(* IEC 61131-3 sources: mp-conveyorbelt/test, 4 files *)

(* ---- ProcessStateAssert.st ---- *)
USING Simatic.Ax.Process;
USING AxUnit.ResultFunctions;
USING System.Strings;
USING Simatic.Ax.Process;

NAMESPACE AxUnit.Assert
    FUNCTION PUBLIC Equal
        VAR_INPUT
            actual : ProcessState;
            expected: ProcessState;
            {CallerFilePath}
            file : WSTRING[1024];
            {CallerLineNumber}
            line : INT;
        END_VAR

        IF actual = expected THEN
            axunit_Succeed();
        ELSE
            axunit_Fail('ProcessState assertion failed', file, line);
        END_IF;

    END_FUNCTION
END_NAMESPACE

(* ---- conveyorbelt-tests.st ---- *)
USING Simatic.Ax.Mp;

NAMESPACE SimaticAxMp

    {TestFixture}
    CLASS Test_SensorInfeed
        {Test}
        METHOD PUBLIC Test_x
            AxUnit.Assert.Equal(expected := 2, actual := 2);
        END_METHOD
        {Test}
        METHOD PUBLIC Test_y
            ; // AxUnit.Assert.Equal(expected := y, actual := x);
        END_METHOD
    END_CLASS

    {TestFixture}
    CLASS Test_SensorWork
        {Test}
        METHOD PUBLIC Test_x
            ; // AxUnit.Assert.Equal(expected := y, actual := x);
        END_METHOD
        {Test}
        METHOD PUBLIC Test_y
            ; // AxUnit.Assert.Equal(expected := y, actual := x);
        END_METHOD
    END_CLASS

    {TestFixture}
    CLASS Test_SensorOutfeed
        {Test}
        METHOD PUBLIC Test_x
            ; // AxUnit.Assert.Equal(expected := y, actual := x);
        END_METHOD
        {Test}
        METHOD PUBLIC Test_y
            ; // AxUnit.Assert.Equal(expected := y, actual := x);
        END_METHOD
    END_CLASS

    {TestFixture}
    CLASS Test_AxisControl
        {Test}
        METHOD PUBLIC Test_x
            ; // AxUnit.Assert.Equal(expected := y, actual := x);
        END_METHOD
        {Test}
        METHOD PUBLIC Test_y
            ; // AxUnit.Assert.Equal(expected := y, actual := x);
        END_METHOD
    END_CLASS

    {TestFixture}
    CLASS Test_ConveyorBelt
        {Test}
        METHOD PUBLIC Test_Init
            ; // AxUnit.Assert.Equal(expected := y, actual := x);
        END_METHOD
        {Test}
        METHOD PUBLIC Test_MoveToSensor_Work_dir1
            ; // AxUnit.Assert.Equal(expected := y, actual := x);
        END_METHOD
        {Test}
        METHOD PUBLIC Test_MoveToSensor_Work_dir0
            ; // AxUnit.Assert.Equal(expected := y, actual := x);
        END_METHOD
        {Test}
        METHOD PUBLIC Test_MoveToSensor_Outfeed_dir1
            ; // AxUnit.Assert.Equal(expected := y, actual := x);
        END_METHOD
        {Test}
        METHOD PUBLIC Test_MoveToSensor_Outfeed_dir0
            ; // AxUnit.Assert.Equal(expected := y, actual := x);
        END_METHOD
        METHOD PUBLIC Test_MoveToSensor_Infeed_dir1
            ; // AxUnit.Assert.Equal(expected := y, actual := x);
        END_METHOD
        {Test}
        METHOD PUBLIC Test_MoveToSensor_Infeed_dir0
            ; // AxUnit.Assert.Equal(expected := y, actual := x);
        END_METHOD

    END_CLASS

END_NAMESPACE

(* ---- conveyors-tests.st ---- *)
USING Simatic.Ax.Mp;

NAMESPACE SimaticAxMp

    {TestFixture}
    CLASS Test_SensorInfeed
        {Test}
        METHOD PUBLIC Test_x
            ; // AxUnit.Assert.Equal(expected := y, actual := x);
        END_METHOD
        {Test}
        METHOD PUBLIC Test_y
            ; // AxUnit.Assert.Equal(expected := y, actual := x);
        END_METHOD
    END_CLASS

    {TestFixture}
    CLASS Test_SensorWork
        {Test}
        METHOD PUBLIC Test_x
            ; // AxUnit.Assert.Equal(expected := y, actual := x);
        END_METHOD
        {Test}
        METHOD PUBLIC Test_y
            ; // AxUnit.Assert.Equal(expected := y, actual := x);
        END_METHOD
    END_CLASS

    {TestFixture}
    CLASS Test_SensorOutfeed
        {Test}
        METHOD PUBLIC Test_x
            ; // AxUnit.Assert.Equal(expected := y, actual := x);
        END_METHOD
        {Test}
        METHOD PUBLIC Test_y
            ; // AxUnit.Assert.Equal(expected := y, actual := x);
        END_METHOD
    END_CLASS

    {TestFixture}
    CLASS Test_AxisControl
        {Test}
        METHOD PUBLIC Test_x
            ; // AxUnit.Assert.Equal(expected := y, actual := x);
        END_METHOD
        {Test}
        METHOD PUBLIC Test_y
            ; // AxUnit.Assert.Equal(expected := y, actual := x);
        END_METHOD
    END_CLASS

    {TestFixture}
    CLASS Test_ConveyorBelt
        {Test}
        METHOD PUBLIC Test_Init
            ; // AxUnit.Assert.Equal(expected := y, actual := x);
        END_METHOD
        {Test}
        METHOD PUBLIC Test_MoveToSensor_Work_dir1
            ; // AxUnit.Assert.Equal(expected := y, actual := x);
        END_METHOD
        {Test}
        METHOD PUBLIC Test_MoveToSensor_Work_dir0
            ; // AxUnit.Assert.Equal(expected := y, actual := x);
        END_METHOD
        {Test}
        METHOD PUBLIC Test_MoveToSensor_Outfeed_dir1
            ; // AxUnit.Assert.Equal(expected := y, actual := x);
        END_METHOD
        {Test}
        METHOD PUBLIC Test_MoveToSensor_Outfeed_dir0
            ; // AxUnit.Assert.Equal(expected := y, actual := x);
        END_METHOD
        METHOD PUBLIC Test_MoveToSensor_Infeed_dir1
            ; // AxUnit.Assert.Equal(expected := y, actual := x);
        END_METHOD
        {Test}
        METHOD PUBLIC Test_MoveToSensor_Infeed_dir0
            ; // AxUnit.Assert.Equal(expected := y, actual := x);
        END_METHOD

    END_CLASS

END_NAMESPACE

(* ---- test.st ---- *)
USING Simatic.Ax.Mp;

NAMESPACE testConveyors

    {TestFixture}
    CLASS testBelt

        VAR PROTECTED
            myBelt : Belt;
        END_VAR

        {Test}
        METHOD PUBLIC test_initBelt
            VAR_TEMP
                beltDataInOut : types.beltData;
            END_VAR

            beltDataInOut.minSpeed := 1000;
            beltDataInOut.maxSpeed := 8000;
            myBelt.setBeltData(beltData := beltDataInOut);

            AxUnit.Assert.Equal(expected := beltDataInOut.minSpeed, actual := myBelt.getBeltData().minSpeed);
            AxUnit.Assert.Equal(expected := beltDataInOut.maxSpeed, actual := myBelt.getBeltData().maxSpeed);
        END_METHOD

        {Test (inSpeed := 5000, outSpeed := 5000)}
        {Test (inSpeed := -100, outSpeed := 0)}
        {Test (inSpeed := 8500, outSpeed := 0)}
        {Test (inSpeed := 3000, outSpeed := 3500)}
        METHOD PUBLIC test_setSpeed
            VAR_INPUT
                inSpeed : INT;
                outSpeed : INT;
            END_VAR
            VAR_TEMP
                result : types.beltData;
            END_VAR

            THIS.test_initBelt();
            myBelt.setSpeedSP(speedSP := inSpeed);
            AxUnit.Assert.Equal(expected := outSpeed, actual := myBelt.getBeltData().speedSP);
        END_METHOD

    END_CLASS

END_NAMESPACE
